{attribute 'linkalways'} 
{attribute 'no_explicit_call' := 'This FB is a CLASS and must be accessed using methods or properties'}
{attribute 'enable_dynamic_creation'}
FUNCTION_BLOCK _Array0to3OfUSINT EXTENDS ArrayDatatypeBase_1D
VAR CONSTANT
	lBound : DINT := 0;
	uBound : DINT := 3;
END_VAR
VAR
	localData : ARRAY [lBound..uBound] OF USINT;
	activeData : REFERENCE TO ARRAY [lBound..uBound] OF USINT REF= localData;
	elements : ARRAY [lBound..uBound] OF _USINT(0);
	baseType : _USINT(0);
END_VAR

PROPERTY PUBLIC Address : PVOID
GET
Address := ADR(activeData);
END_GET
END_PROPERTY

PROPERTY PUBLIC BaseDatatype : I_Datatype
GET
BaseDatatype := baseType;
END_GET
END_PROPERTY

METHOD PUBLIC ClearReference
VAR_INPUT
END_VAR
activeData REF= localData;
SetElementReference();
END_METHOD

METHOD PUBLIC Clone : I_Datatype
VAR
    pClone : POINTER TO _Array0to3OfUSINT;
END_VAR
pClone := __NEW(_Array0to3OfUSINT());
pClone^.Value := Value;
Clone := pClone^;
END_METHOD

METHOD FB_init : BOOL
VAR_INPUT
	bInitRetains : BOOL; // if TRUE, the retain variables are initialized (warm start / cold start)
	bInCopyCode : BOOL;  // if TRUE, the instance afterwards gets moved into the copy code (online change)
END_VAR
SetElementReference();
END_METHOD

METHOD PUBLIC MakeReferenceTo
VAR_INPUT
	ReferenceTarget : REFERENCE TO ARRAY [lBound..uBound] OF USINT;
END_VAR
activeData REF= ReferenceTarget;
SetElementReference();
END_METHOD

METHOD PROTECTED OnSerializeArrayValues
VAR_INPUT
	Serializer : I_Serializer;
END_VAR
VAR
	i : DINT;
END_VAR
FOR i := lBound TO uBound DO
	elements[i].SerializeWith(Serializer);
END_FOR
END_METHOD

METHOD PROTECTED SetElementReference
VAR_INPUT
END_VAR
VAR
	i : DINT;
END_VAR
FOR i := lBound TO uBound DO
	elements[i].MakeReferenceTo(activeData[i]);
END_FOR
END_METHOD

PROPERTY PUBLIC Size : UDINT
GET
Size := SIZEOF(activeData);
END_GET
END_PROPERTY

METHOD PROTECTED TryDeserializeArrayValues : BOOL
VAR_INPUT
	Deserializer : I_Deserializer;
	Feedback : I_DeserializerFeedback;
END_VAR
VAR
	enumerator : I_DeserializerArrayForwardEnumerator;
	i : DINT;
END_VAR
enumerator := Deserializer.GetArrayEnumerator();
i := lBound;

WHILE enumerator.MoveNext() AND i <= uBound DO
	
	IF NOT elements[i].TryDeserializeFrom(enumerator.Current, Feedback) THEN
		EXIT;
	END_IF
	i := i + 1;

END_WHILE
enumerator.Dispose();
END_METHOD

METHOD PUBLIC TryGetElementAsDatatypeByIndex : BOOL
VAR_INPUT
	Index : DINT;
	Destination : REFERENCE TO I_Datatype;
END_VAR
IF Index < lbound OR Index > ubound THEN
	RETURN;
END_IF

Destination := elements[Index];
TryGetElementAsDatatypeByIndex := TRUE;
END_METHOD

METHOD PUBLIC TryGetLowerBound : BOOL
VAR_INPUT
	Dimention : UDINT;
	Destination : REFERENCE TO DINT;
END_VAR
IF Dimention = 1 THEN
	Destination := lBound;
	TryGetLowerBound := TRUE;
END_IF
END_METHOD

METHOD PUBLIC TryGetUpperBound : BOOL
VAR_INPUT
	Dimention : UDINT;
	Destination : REFERENCE TO DINT;
END_VAR
IF Dimention = 1 THEN
	Destination := uBound;
	TryGetUpperBound := TRUE;
END_IF
END_METHOD

METHOD TryMakeReferenceTo : BOOL
VAR_INPUT
	Target : I_Datatype;
END_VAR
VAR
	targetAsArray : I_ArrayDatatype;
	pTargetData : POINTER TO ARRAY [lBound..uBound] OF USINT;
END_VAR
IF NOT Target.TryResolveAsArrayDatatype(targetAsArray) THEN
	RETURN;
END_IF

IF NOT (targetAsArray.Identifier = Identifier) THEN
	RETURN;
END_IF

pTargetData := Target.Address;
activeData REF= pTargetData^;
SetElementReference();
TryMakeReferenceTo := TRUE;
END_METHOD

PROPERTY PUBLIC Value : REFERENCE TO ARRAY [lBound..uBound] OF USINT;
GET
Value ref= activeData;
END_GET
END_PROPERTY

END_FUNCTION_BLOCK

(* stored: Version 1.1.0.1, ProductVersion 3.1.4024.13
   POU _Array0to3OfUSINT: Id {998419e9-395b-0923-3713-ec2e733a5a4d}, SpecialFunc None
   Folder Core: Id {210ff53f-4c69-0341-0be1-1239ec29a67a}
   Folder Constructor: Id {c0c78977-35bc-0f81-0925-5acd6f13500f}
   Folder Protected: Id {db9961d7-cb56-0c68-2513-6b3b080455b8}
   Folder Customize: Id {b5a16647-f12d-0ee0-111d-0cdce096d9a5}
   Property Address: Id {b4976d00-638c-0c74-34cb-0f67febcdee9}
   Get Get: Id {25996113-d003-01de-2200-e3b5ab278e12}
   Property BaseDatatype: Id {c523f7d2-05f4-036a-0d44-41f49e3392c0}
   Get Get: Id {a07cdb84-c2d4-0daf-3904-85eb2bca26ac}
   Method ClearReference: Id {271a07b5-6707-0603-19a1-5d909514ca24}
   Method Clone: Id {5822c416-8e40-0df0-13f4-09d280524f87}
   Method FB_init: Id {67c3551e-310f-0ac0-07ec-6bbf2f73d905}
   Method MakeReferenceTo: Id {11781d7d-20af-078a-1d1b-bf97a1eb4052}
   Method OnSerializeArrayValues: Id {efd000df-57ea-053d-00b6-99ff33dd074e}
   Method SetElementReference: Id {0e4802de-10a2-0543-232d-c0bb5c55b393}
   Property Size: Id {6e2fe7ab-b384-0d9a-3ad5-d38dfc008b7f}
   Get Get: Id {f91016aa-f7f5-0523-0fad-23ee28453836}
   Method TryDeserializeArrayValues: Id {abae1611-6da5-0d7f-1ec7-91cf6a081d08}
   Method TryGetElementAsDatatypeByIndex: Id {38485966-f18e-0521-06a2-3028c6f47473}
   Method TryGetLowerBound: Id {b84601a1-d89e-053d-0d93-daa3a29ec307}
   Method TryGetUpperBound: Id {ec667316-4c72-03a6-02c0-df56c9dcd4b5}
   Method TryMakeReferenceTo: Id {231ee423-a3fc-0046-0fb3-e0d951dc5afd}
   Property Value: Id {8fe15983-577f-07a4-29c1-0f3b5ad811fd}
   Get Get: Id {c99b89ca-7be2-064a-0fef-f32118c955e5} *)
